KUKA KRL program: tet.src, tet.dat

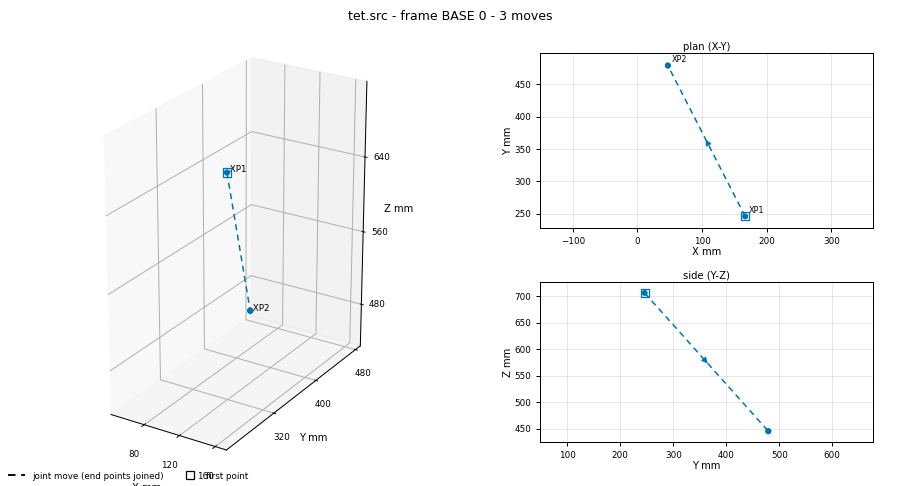
[picture p0: tool path of tet.src in frame BASE 0, 3 of 3 moves have a stored position in this frame; points joined in program order, loops and branches not executed]
--- tet.src ---
&ACCESS RVO
&REL 9
&PARAM EDITMASK = *
&PARAM TEMPLATE = C:\KRC\Roboter\Template\vorgabe
&PARAM DISKPATH = KRC:\R1\Program\fon022
DEF tet( )
;FOLD INI;%{PE}
  ;FOLD BASISTECH INI
    GLOBAL INTERRUPT DECL 3 WHEN $STOPMESS==TRUE DO IR_STOPM ( )
    INTERRUPT ON 3
    BAS (#INITMOV,0 )
  ;ENDFOLD (BASISTECH INI)
  ;FOLD USER INI
    ;Make your modifications here

  ;ENDFOLD (USER INI)
;ENDFOLD (INI)


;FOLD PTP P1 Vel=100 % PDAT1 Tool[1] Base[0] ;%{PE}
;FOLD Parameters ;%{h}
;Params IlfProvider=kukaroboter.basistech.inlineforms.movement.old; Kuka.IsGlobalPoint=False; Kuka.PointName=P1; Kuka.BlendingEnabled=False; Kuka.MoveDataPtpName=PDAT1; Kuka.VelocityPtp=100; Kuka.CurrentCDSetIndex=0; Kuka.MovementParameterFieldEnabled=True; IlfCommand=PTP
;ENDFOLD
$BWDSTART = FALSE
PDAT_ACT = PPDAT1
FDAT_ACT = FP1
BAS(#PTP_PARAMS, 100.0)
SET_CD_PARAMS (0)
PTP XP1
;ENDFOLD

;FOLD SPTP P2 Vel=100 % PDAT2 Tool[1] Base[0] ;%{PE}
;FOLD Parameters ;%{h}
;Params IlfProvider=kukaroboter.basistech.inlineforms.movement.spline; Kuka.IsGlobalPoint=False; Kuka.PointName=P2; Kuka.BlendingEnabled=False; Kuka.MoveDataPtpName=PDAT2; Kuka.VelocityPtp=100; Kuka.VelocityFieldEnabled=True; Kuka.ColDetectFieldEnabled=True; Kuka.CurrentCDSetIndex=0; Kuka.MovementParameterFieldEnabled=True; IlfCommand=SPTP
;ENDFOLD
SPTP XP2 WITH $VEL_AXIS[1] = SVEL_JOINT(100.0), $TOOL = STOOL2(FP2), $BASE = SBASE(FP2.BASE_NO), $IPO_MODE = SIPO_MODE(FP2.IPO_FRAME), $LOAD = SLOAD(FP2.TOOL_NO), $ACC_AXIS[1] = SACC_JOINT(PPDAT2), $APO = SAPO_PTP(PPDAT2), $GEAR_JERK[1] = SGEAR_JERK(PPDAT2), $COLLMON_TOL_PRO[1] = USE_CM_PRO_VALUES(0)
;ENDFOLD
;FOLD SPTP P3 Vel=100 % PDAT3 Tool[1] Base[0] ;%{PE}
;FOLD Parameters ;%{h}
;Params IlfProvider=kukaroboter.basistech.inlineforms.movement.spline; Kuka.IsGlobalPoint=False; Kuka.PointName=P3; Kuka.BlendingEnabled=False; Kuka.MoveDataPtpName=PDAT3; Kuka.VelocityPtp=100; Kuka.VelocityFieldEnabled=True; Kuka.ColDetectFieldEnabled=True; Kuka.CurrentCDSetIndex=0; Kuka.MovementParameterFieldEnabled=True; IlfCommand=SPTP
;ENDFOLD
SPTP XP3 WITH $VEL_AXIS[1] = SVEL_JOINT(100.0), $TOOL = STOOL2(FP3), $BASE = SBASE(FP3.BASE_NO), $IPO_MODE = SIPO_MODE(FP3.IPO_FRAME), $LOAD = SLOAD(FP3.TOOL_NO), $ACC_AXIS[1] = SACC_JOINT(PPDAT3), $APO = SAPO_PTP(PPDAT3), $GEAR_JERK[1] = SGEAR_JERK(PPDAT3), $COLLMON_TOL_PRO[1] = USE_CM_PRO_VALUES(0)
;ENDFOLD
END

--- tet.dat ---
&ACCESS RVO
&REL 9
&PARAM EDITMASK = *
&PARAM TEMPLATE = C:\KRC\Roboter\Template\vorgabe
&PARAM DISKPATH = KRC:\R1\Program\fon022
DEFDAT  TET
;FOLD EXTERNAL DECLARATIONS;%{PE}%MKUKATPBASIS,%CEXT,%VCOMMON,%P
;FOLD BASISTECH EXT;%{PE}%MKUKATPBASIS,%CEXT,%VEXT,%P
EXT  BAS (BAS_COMMAND  :IN,REAL  :IN )
DECL INT SUCCESS
;ENDFOLD (BASISTECH EXT)
;FOLD USER EXT;%{E}%MKUKATPUSER,%CEXT,%VEXT,%P
;Make your modifications here

;ENDFOLD (USER EXT)
;ENDFOLD (EXTERNAL DECLARATIONS)
DECL E6POS XP1={X 166.719391,Y 245.978134,Z 706.313232,A 44.8099,B -62.6632729,C -166.082458,S 2,T 11,E1 0.0,E2 0.0,E3 0.0,E4 0.0,E5 0.0,E6 0.0}
DECL FDAT FP1={TOOL_NO 1,BASE_NO 0,IPO_FRAME #BASE,POINT2[] " "}
DECL PDAT PPDAT1={VEL 100.000,ACC 100.000,APO_DIST 500.000,APO_MODE #CDIS,GEAR_JERK 100.000,EXAX_IGN 0}
DECL MODULEPARAM_T LAST_TP_PARAMS={PARAMS[] "Kuka.PointName=P3; Kuka.FrameData.base_no=0; Kuka.FrameData.tool_no=1; Kuka.FrameData.ipo_frame=#BASE; Kuka.isglobalpoint=False; Kuka.MoveDataPtpName=PDAT3; Kuka.MovementDataPdat.apo_mode=#CDIS; Kuka.MovementDataPdat.apo_dist=500; Kuka.MovementData.vel=100; Kuka.MovementData.acc=100; Kuka.MovementData.exax_ign=0; Kuka.VelocityPtp=100; Kuka.BlendingEnabled=False; Kuka.APXEnabled=False; Kuka.CurrentCDSetIndex=0; Kuka.VelocityFieldEnabled=True; Kuka.ColDetectFieldEnabled=True; Kuka.MovementParameterFieldEnabled=True; Kuka.IsAngleEnabled=False; Kuka.FrameData.point2="}
DECL E6POS XP2={X 47.1443825,Y 479.281,Z 445.467926,A 85.1207809,B -0.646964312,C -176.616211,S 2,T 11,E1 0.0,E2 0.0,E3 0.0,E4 0.0,E5 0.0,E6 0.0}
DECL FDAT FP2={TOOL_NO 1,BASE_NO 0,IPO_FRAME #BASE,POINT2[] " "}
DECL PDAT PPDAT2={VEL 100.000,ACC 100.000,APO_DIST 500.000,APO_MODE #CDIS,GEAR_JERK 100.000,EXAX_IGN 0}
DECL E6POS XP3={X 47.1396065,Y 479.282166,Z 445.460449,A 7.13081503,B 3.17615676,C -178.665726,S 2,T 11,E1 0.0,E2 0.0,E3 0.0,E4 0.0,E5 0.0,E6 0.0}
DECL FDAT FP3={TOOL_NO 1,BASE_NO 0,IPO_FRAME #BASE,POINT2[] " "}
DECL PDAT PPDAT3={VEL 100.000,ACC 100.000,APO_DIST 500.000,APO_MODE #CDIS,GEAR_JERK 100.000,EXAX_IGN 0}
ENDDAT
